FUNCTION_BLOCK UDINT2REAL (* Basic Function Block Type *)
  (* Standard: 61499-2 *)
  (* Version 0.0, 7/4/2026, Schneider Electric, Template *)
  PACKAGE SE.Nereda;
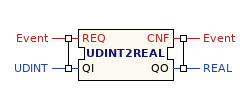
  EVENT_INPUT
    REQ WITH QI; (* Normal Execution Request *)
  END_EVENT
  EVENT_OUTPUT
    CNF WITH QO; (* Execution Confirmation *)
  END_EVENT
  VAR_INPUT
    QI : UDINT; (* Input event qualifier *)
  END_VAR
  VAR_OUTPUT
    QO : REAL; (* Output event qualifier *)
  END_VAR
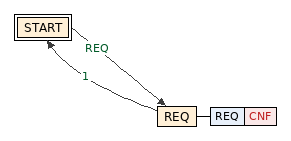
  EC_STATES
    START; (* Initial State *)
    REQ : REQ -> CNF; (* Normal execution *)
  END_STATES
  EC_TRANSITIONS
    START TO REQ := REQ;
    REQ TO START := 1;
  END_TRANSITIONS
  ALGORITHM REQ IN ST: (* Normally executed algorithm *)
;
QO := UDINT_TO_REAL(QI);
  END_ALGORITHM
END_FUNCTION_BLOCK
